RoboDK station: Übung3.rdk

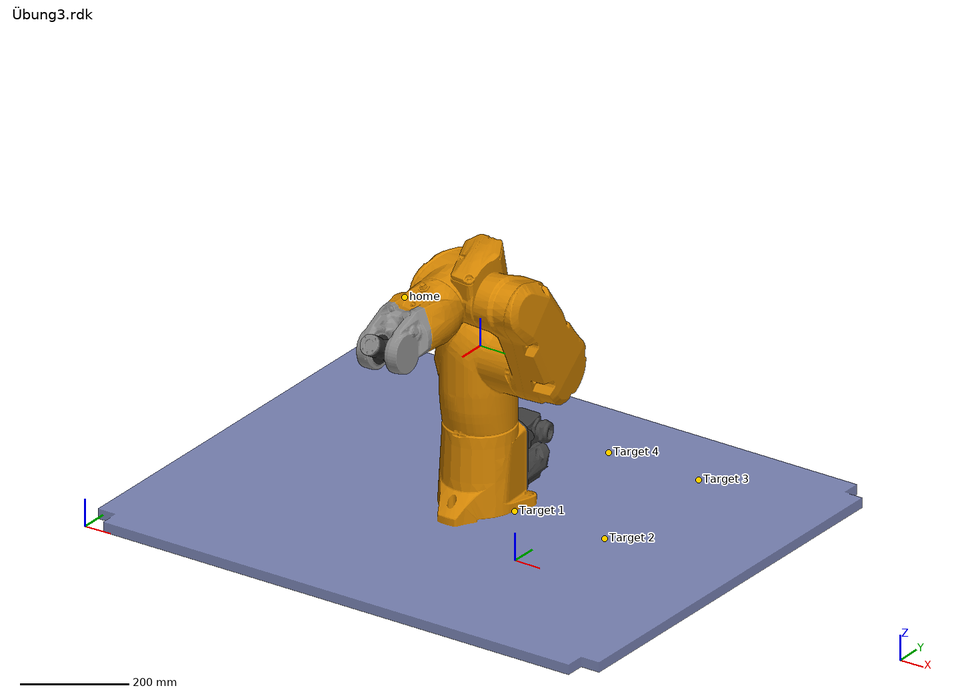
[picture v0: the station drawn from its stored meshes, robots at their saved joint values, targets as dots, program paths as lines]
Station Übung3 (saved by RoboDK 5.6.9). Poses are relative to the parent item; angles as X-Y-Z fixed-axis rotations.
  - frame world at (0, 0, 0) mm
    - frame Staubli TX2-40 Base at (560, 460, 340) mm, rotated rx 0 ry 0 rz -90 deg
      - robot Staubli TX2-40: 6 axes, payload 2 kg, reach 515 mm, repeatability 0.02 mm, weight 29 kg
          modified DH rows (alpha deg, a mm, theta deg, d mm): 0, 0, 0, 320; -90, 0, -90, 35; 0, 225, -90, 0; -90, 0, 0, 225; 90, 0, 0, 0; -90, 0, 180, 65
          base shift (0, 0, -320) mm
          joint limits [-180, -125, -138, -270, -120, -270] to [180, 125, 138, 270, 133.5, 270]; home [0, 0, 90, 0, 0, 0]; saved at [1.45, 37.3, 61.21, 6.53, -40.27, 0]
    - object Arbeitsflaeche_geteilt at (0, 0, 0) mm, size 1120 x 920 x 20 mm, geometry from Arbeitsflaeche_geteilt.iges
    - object Arbeitsflaeche_komplett at (0, 0, 0) mm, size 1120 x 920 x 20 mm, geometry from Arbeitsflaeche_komplett.IGS
    - object Zelle at (0, 0, 0) mm, rotated rx 90 ry 0 rz -90 deg, size 1120 x 1947.8 x 1200 mm, geometry from Zelle.stp
    - target home (Cartesian target) at (595, 170, 565) mm, rotated rx 0 ry 90 rz -90 deg; joints [0, 0, 90, 0, 0, 0] of Staubli TX2-40
    - frame cuboid at (750, 300, 20) mm
      - object cuboid at (0, 0, 0) mm, size 200 x 300 x 100 mm, geometry from cuboid.iges
      - target Target 1 (Cartesian target) at (0, 0, 100) mm, rotated rx 180 ry 0 rz 90 deg; joints [41.799, 72.462, 99.522, 0, 8.016, 41.799] of Staubli TX2-40
      - target Target 2 (Cartesian target) at (200, 0, 100) mm, rotated rx -180 ry 0 rz -180 deg; joints [62.931, 104.549, 11.407, 180, -64.044, 152.931] of Staubli TX2-40
      - target Target 3 (Cartesian target) at (200, 300, 100) mm, rotated rx 180 ry 0 rz -90 deg; joints [-65.408, -122.041, 22.929, 0, -80.888, 114.592] of Staubli TX2-40
      - target Target 4 (Cartesian target) at (0, 300, 100) mm, rotated rx 180 ry 0 rz 0 deg; joints [117.856, 72.096, 102.985, 0, 4.92, 207.856] of Staubli TX2-40
  - Python program Prog3 (listed below)

--- Python program Prog3 ---
# Type help("robodk.robolink") or help("robodk.robomath") for more information
# Press F5 to run the script
# Documentation: https://robodk.com/doc/en/RoboDK-API.html
# Reference:     https://robodk.com/doc/en/PythonAPI/robodk.html
# Note: It is not required to keep a copy of this file, your Python script is saved with your RDK project
from robodk.robolink import *      # RoboDK API
from robodk.robomath import *    # Robot link toolbox

# Link to RoboDK
RDK = Robolink()

robot = RDK.Item('Staubli TX2-40')

world = RDK.Item('world')
home = RDK.Item('home')
cuboid = RDK.Item('cuboid')
target1 = RDK.Item('Target 1')
target2 = RDK.Item('Target 2')
target3 = RDK.Item('Target 3')
target4 = RDK.Item('Target 4')

print('start')

robot.setAccelerationJoints(150)
robot.setSpeedJoints(150)

#
robot.setSpeed(20, 20, 150, 150)

robot.setPoseFrame(world)
robot.MoveJ(home)
robot.setPoseFrame(cuboid)
robot.MoveJ(target1)
robot.MoveL(target2)
robot.MoveL(target3)
robot.MoveL(target4)
robot.setPoseFrame(world)
robot.MoveJ(home)

print('end')
